DATA_BLOCK "DB"
{ S7_Optimized_Access := 'false' }
    VAR
        S_an_output: DINT;
        S_a_wire: BOOL;
        S_data: REAL;
        avalue: DINT;
        flag: BOOL;
        measurement: REAL;
        firstRun: BOOL;
    END_VAR
BEGIN
    firstRun := TRUE;
END_DATA_BLOCK
